PROGRAM prgPerData
VAR
	fbPerData			: FB_WritePersistentData_CX81xx;
END_VAR

fbPerData(
	eSaveModeData:= eUSVSaveMode.eSaveWhenPowerfail, 
	bLoadPersistentDataOk=> , 
	bPowerFailDetect=> , 
	bError=> , 
	bySaveProcess=> , 
	dwStorageLast24h=> , 
	udiErrorCode=> );

END_PROGRAM

(* stored: Version 1.1.0.1, ProductVersion 3.1.4024.9
   POU prgPerData: Id {99777527-37bb-4f53-af68-43827fbda431}, SpecialFunc None *)
